TYPE ST_Component :
STRUCT
	bPause:				BOOL;
    bHold:				BOOL;
	bComplete:			BOOL;
END_STRUCT
END_TYPE

(* stored: Version 1.1.0.1
   DUT ST_Component: Id {f31558f2-ea02-4195-a5dc-8f2035d5f64a} *)
